VISUALIZATION VISU_State_green_red  // 12x17
VAR_IN_OUT
	state : BOOL;
END_VAR
    Ellipse (0,5 10x10), colour toggle: state
END_VISUALIZATION

(* stored: Version 1.1.0.1, ProductVersion 3.1.0.36
   Visu VISU_State_green_red: Id {92cb3104-567e-4826-9a75-27d29851d0c5} *)
